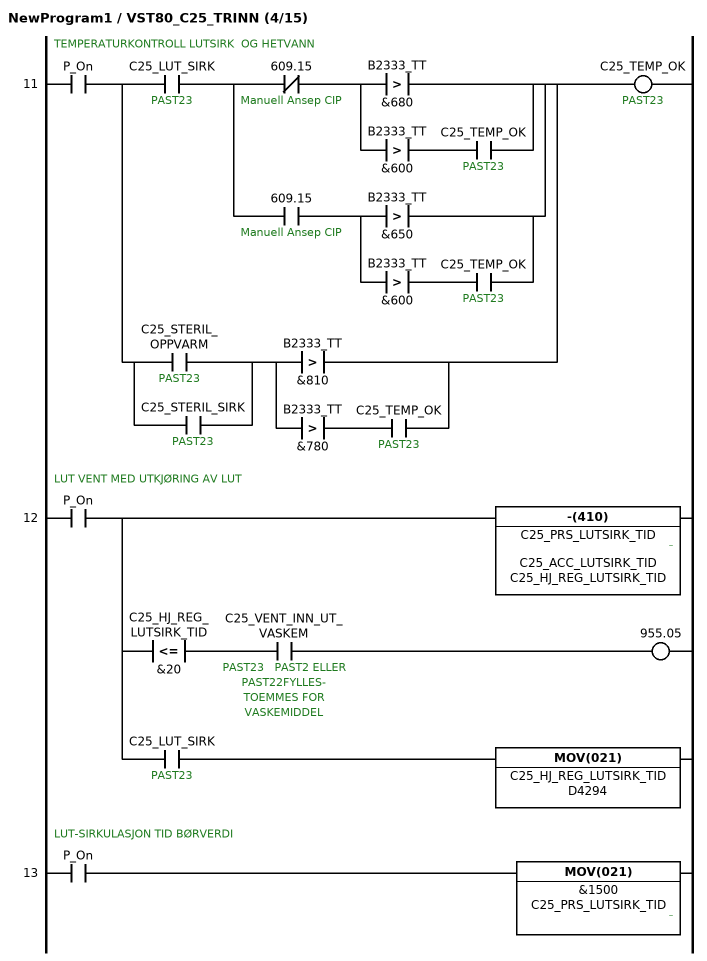
; [picture p456: NewProgram1 / VST80_C25_TRINN, rungs 11-13]
; rung 11: TEMPERATURKONTROLL LUTSIRK  OG HETVANN
LD P_On
LD C25_LUT_SIRK  ; PAST23
LDNOT 609.15  ; Manuell Ansep CIP
LD>(320) B2333_TT &680
LD>(320) B2333_TT &600
AND C25_TEMP_OK  ; PAST23
ORLD
ANDLD
LD 609.15  ; Manuell Ansep CIP
LD>(320) B2333_TT &650
LD>(320) B2333_TT &600
AND C25_TEMP_OK  ; PAST23
ORLD
ANDLD
ORLD
ANDLD
LD C25_STERIL_OPPVARM  ; PAST23
OR C25_STERIL_SIRK  ; PAST23
LD>(320) B2333_TT &810
LD>(320) B2333_TT &780
AND C25_TEMP_OK  ; PAST23
ORLD
ANDLD
ORLD
ANDLD
OUT C25_TEMP_OK  ; PAST23
; rung 12: LUT VENT MED UTKJØRING AV LUT
LD P_On
OUT TR0
-(410) C25_PRS_LUTSIRK_TID C25_ACC_LUTSIRK_TID C25_HJ_REG_LUTSIRK_TID  ; ¨
AND<=(315) C25_HJ_REG_LUTSIRK_TID &20
AND C25_VENT_INN_UT_VASKEM  ; PAST23   PAST2 ELLER PAST22FYLLES-TOEMMES FOR VASKEMIDDEL
OUT 955.05
LD TR0
AND C25_LUT_SIRK  ; PAST23
MOV(021) C25_HJ_REG_LUTSIRK_TID D4294
; rung 13: LUT-SIRKULASJON TID BØRVERDI
LD P_On
MOV(021) &1500 C25_PRS_LUTSIRK_TID  ; ¨

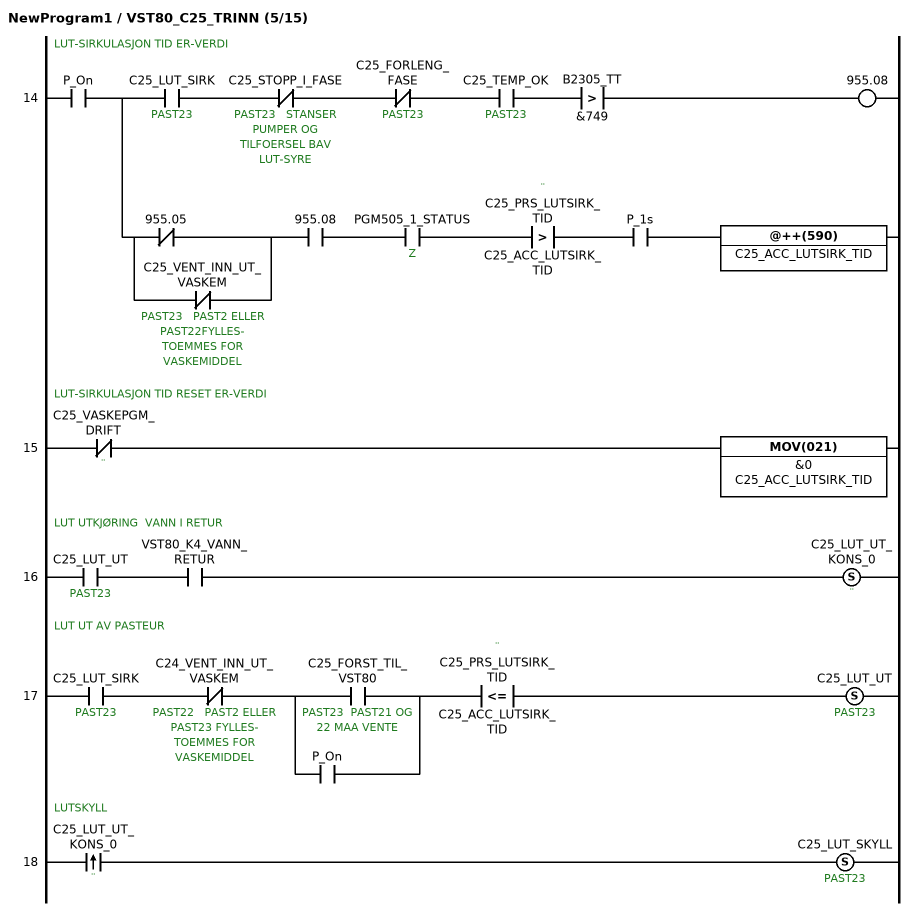
; rung 14: LUT-SIRKULASJON TID ER-VERDI
LD P_On
OUT TR0
AND C25_LUT_SIRK  ; PAST23
ANDNOT C25_STOPP_I_FASE  ; PAST23   STANSER PUMPER OG TILFOERSEL BAV LUT-SYRE
ANDNOT C25_FORLENG_FASE  ; PAST23
AND C25_TEMP_OK  ; PAST23
AND>(320) B2305_TT &749
OUT 955.08
LD TR0
LDNOT 955.05
ORNOT C25_VENT_INN_UT_VASKEM  ; PAST23   PAST2 ELLER PAST22FYLLES-TOEMMES FOR VASKEMIDDEL
ANDLD
AND 955.08
AND PGM505_1_STATUS  ; Z
AND>(320) C25_PRS_LUTSIRK_TID C25_ACC_LUTSIRK_TID  ; ¨
AND P_1s
@++(590) C25_ACC_LUTSIRK_TID
; rung 15: LUT-SIRKULASJON TID RESET ER-VERDI
LDNOT C25_VASKEPGM_DRIFT  ; ¨
MOV(021) &0 C25_ACC_LUTSIRK_TID
; rung 16: LUT UTKJØRING  VANN I RETUR
LD C25_LUT_UT  ; PAST23
AND VST80_K4_VANN_RETUR
SET C25_LUT_UT_KONS_0  ; ¨
; rung 17: LUT UT AV PASTEUR
LD C25_LUT_SIRK  ; PAST23
ANDNOT C24_VENT_INN_UT_VASKEM  ; PAST22   PAST2 ELLER PAST23 FYLLES-TOEMMES FOR VASKEMIDDEL
LD C25_FORST_TIL_VST80  ; PAST23  PAST21 OG 22 MAA VENTE
OR P_On
ANDLD
AND<=(315) C25_PRS_LUTSIRK_TID C25_ACC_LUTSIRK_TID  ; ¨
SET C25_LUT_UT  ; PAST23
; rung 18: LUTSKYLL
@LD C25_LUT_UT_KONS_0  ; ¨
SET C25_LUT_SKYLL  ; PAST23

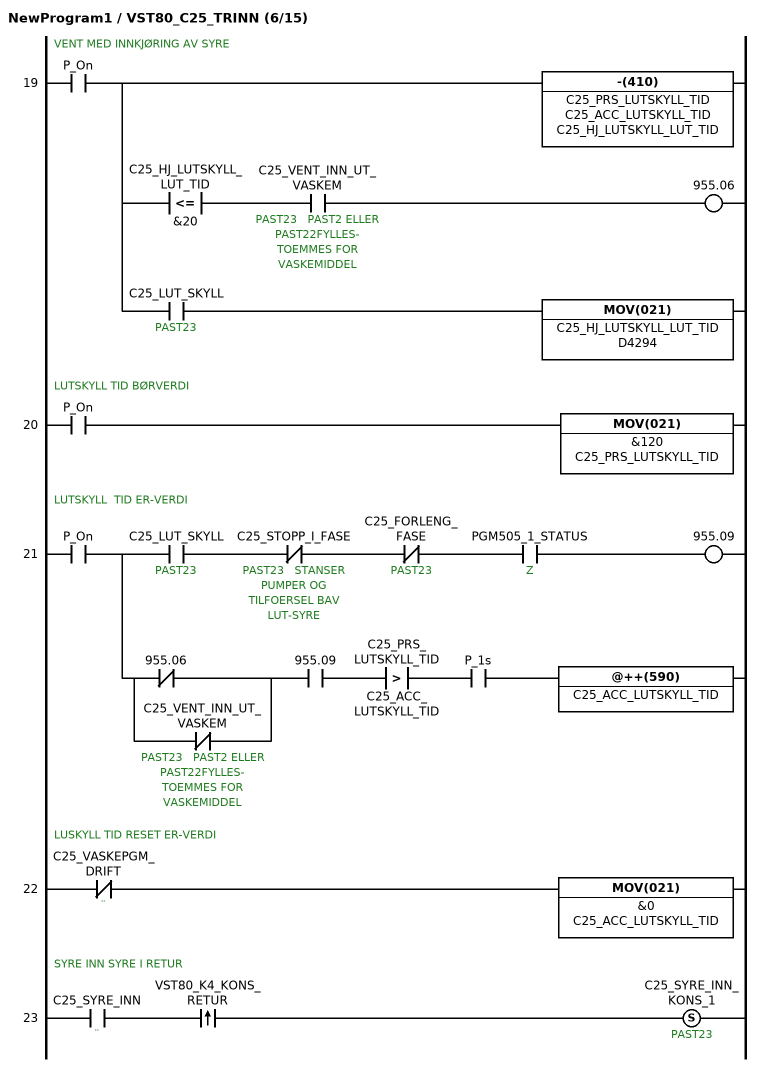
; rung 19: VENT MED INNKJØRING AV SYRE
LD P_On
OUT TR0
-(410) C25_PRS_LUTSKYLL_TID C25_ACC_LUTSKYLL_TID C25_HJ_LUTSKYLL_LUT_TID
AND<=(315) C25_HJ_LUTSKYLL_LUT_TID &20
AND C25_VENT_INN_UT_VASKEM  ; PAST23   PAST2 ELLER PAST22FYLLES-TOEMMES FOR VASKEMIDDEL
OUT 955.06
LD TR0
AND C25_LUT_SKYLL  ; PAST23
MOV(021) C25_HJ_LUTSKYLL_LUT_TID D4294
; rung 20: LUTSKYLL TID BØRVERDI
LD P_On
MOV(021) &120 C25_PRS_LUTSKYLL_TID
; rung 21: LUTSKYLL  TID ER-VERDI
LD P_On
OUT TR0
AND C25_LUT_SKYLL  ; PAST23
ANDNOT C25_STOPP_I_FASE  ; PAST23   STANSER PUMPER OG TILFOERSEL BAV LUT-SYRE
ANDNOT C25_FORLENG_FASE  ; PAST23
AND PGM505_1_STATUS  ; Z
OUT 955.09
LD TR0
LDNOT 955.06
ORNOT C25_VENT_INN_UT_VASKEM  ; PAST23   PAST2 ELLER PAST22FYLLES-TOEMMES FOR VASKEMIDDEL
ANDLD
AND 955.09
AND>(320) C25_PRS_LUTSKYLL_TID C25_ACC_LUTSKYLL_TID
AND P_1s
@++(590) C25_ACC_LUTSKYLL_TID
; rung 22: LUSKYLL TID RESET ER-VERDI
LDNOT C25_VASKEPGM_DRIFT  ; ¨
MOV(021) &0 C25_ACC_LUTSKYLL_TID
; rung 23: SYRE INN SYRE I RETUR
LD C25_SYRE_INN  ; ¨
@AND VST80_K4_KONS_RETUR
SET C25_SYRE_INN_KONS_1  ; PAST23

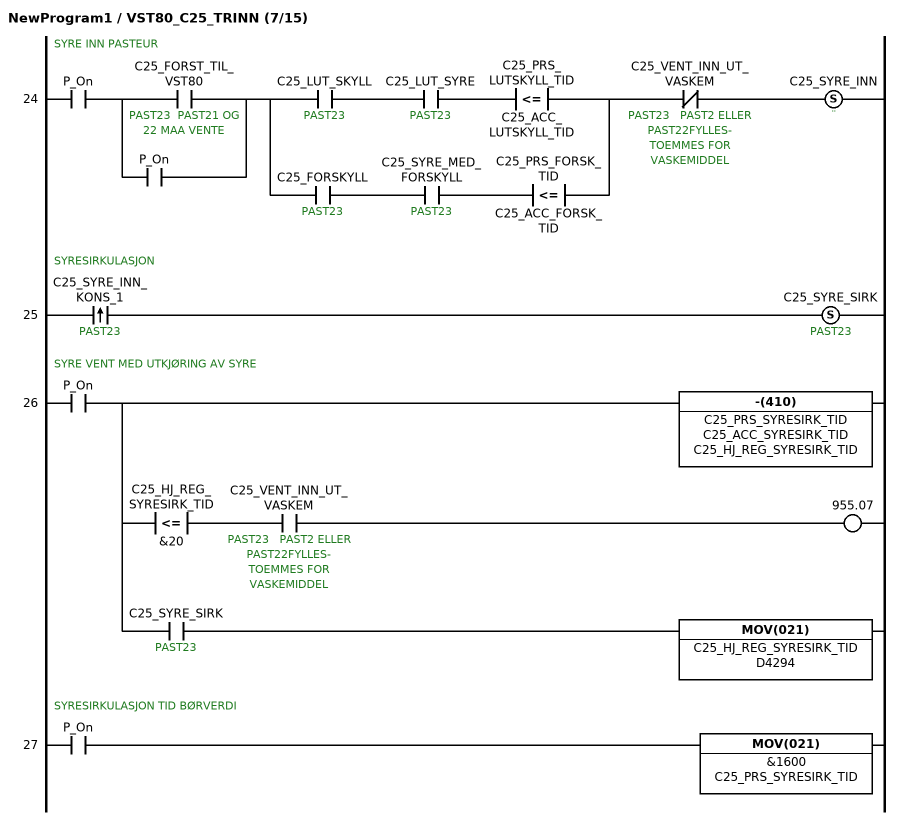
; rung 24: SYRE INN PASTEUR
LD P_On
LD C25_FORST_TIL_VST80  ; PAST23  PAST21 OG 22 MAA VENTE
OR P_On
ANDLD
LD C25_LUT_SKYLL  ; PAST23
AND C25_LUT_SYRE  ; PAST23
AND<=(315) C25_PRS_LUTSKYLL_TID C25_ACC_LUTSKYLL_TID
LD C25_FORSKYLL  ; PAST23
AND C25_SYRE_MED_FORSKYLL  ; PAST23
AND<=(315) C25_PRS_FORSK_TID C25_ACC_FORSK_TID
ORLD
ANDLD
ANDNOT C25_VENT_INN_UT_VASKEM  ; PAST23   PAST2 ELLER PAST22FYLLES-TOEMMES FOR VASKEMIDDEL
SET C25_SYRE_INN  ; ¨
; rung 25: SYRESIRKULASJON
@LD C25_SYRE_INN_KONS_1  ; PAST23
SET C25_SYRE_SIRK  ; PAST23
; rung 26: SYRE VENT MED UTKJØRING AV SYRE
LD P_On
OUT TR0
-(410) C25_PRS_SYRESIRK_TID C25_ACC_SYRESIRK_TID C25_HJ_REG_SYRESIRK_TID
AND<=(315) C25_HJ_REG_SYRESIRK_TID &20
AND C25_VENT_INN_UT_VASKEM  ; PAST23   PAST2 ELLER PAST22FYLLES-TOEMMES FOR VASKEMIDDEL
OUT 955.07
LD TR0
AND C25_SYRE_SIRK  ; PAST23
MOV(021) C25_HJ_REG_SYRESIRK_TID D4294
; rung 27: SYRESIRKULASJON TID BØRVERDI
LD P_On
MOV(021) &1600 C25_PRS_SYRESIRK_TID

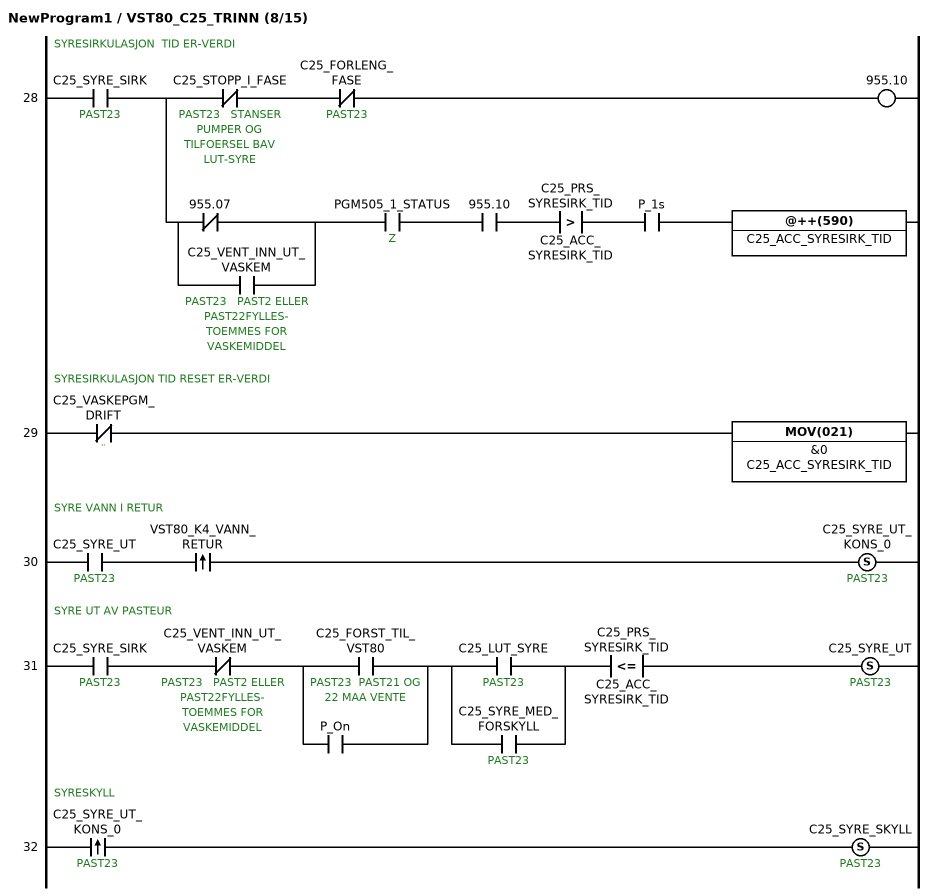
; rung 28: SYRESIRKULASJON  TID ER-VERDI
LD C25_SYRE_SIRK  ; PAST23
OUT TR0
ANDNOT C25_STOPP_I_FASE  ; PAST23   STANSER PUMPER OG TILFOERSEL BAV LUT-SYRE
ANDNOT C25_FORLENG_FASE  ; PAST23
OUT 955.10
LD TR0
LDNOT 955.07
OR C25_VENT_INN_UT_VASKEM  ; PAST23   PAST2 ELLER PAST22FYLLES-TOEMMES FOR VASKEMIDDEL
ANDLD
AND PGM505_1_STATUS  ; Z
AND 955.10
AND>(320) C25_PRS_SYRESIRK_TID C25_ACC_SYRESIRK_TID
AND P_1s
@++(590) C25_ACC_SYRESIRK_TID
; rung 29: SYRESIRKULASJON TID RESET ER-VERDI
LDNOT C25_VASKEPGM_DRIFT  ; ¨
MOV(021) &0 C25_ACC_SYRESIRK_TID
; rung 30: SYRE VANN I RETUR
LD C25_SYRE_UT  ; PAST23
@AND VST80_K4_VANN_RETUR
SET C25_SYRE_UT_KONS_0  ; PAST23
; rung 31: SYRE UT AV PASTEUR
LD C25_SYRE_SIRK  ; PAST23
ANDNOT C25_VENT_INN_UT_VASKEM  ; PAST23   PAST2 ELLER PAST22FYLLES-TOEMMES FOR VASKEMIDDEL
LD C25_FORST_TIL_VST80  ; PAST23  PAST21 OG 22 MAA VENTE
OR P_On
ANDLD
LD C25_LUT_SYRE  ; PAST23
OR C25_SYRE_MED_FORSKYLL  ; PAST23
ANDLD
AND<=(315) C25_PRS_SYRESIRK_TID C25_ACC_SYRESIRK_TID
SET C25_SYRE_UT  ; PAST23
; rung 32: SYRESKYLL
@LD C25_SYRE_UT_KONS_0  ; PAST23
SET C25_SYRE_SKYLL  ; PAST23

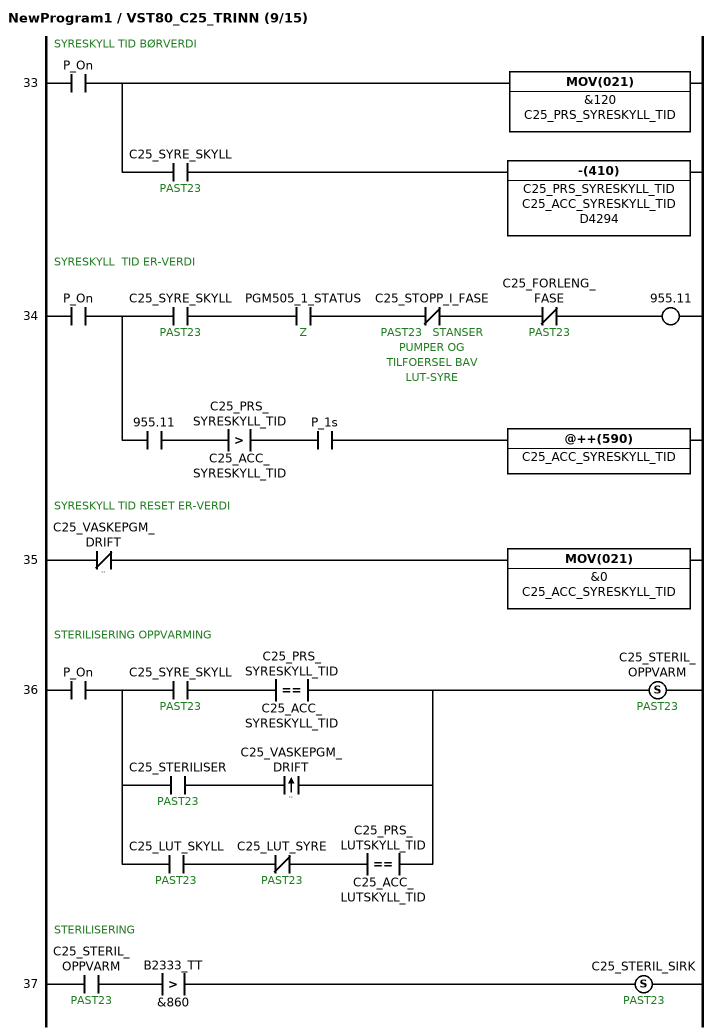
; rung 33: SYRESKYLL TID BØRVERDI
LD P_On
MOV(021) &120 C25_PRS_SYRESKYLL_TID
AND C25_SYRE_SKYLL  ; PAST23
-(410) C25_PRS_SYRESKYLL_TID C25_ACC_SYRESKYLL_TID D4294
; rung 34: SYRESKYLL  TID ER-VERDI
LD P_On
OUT TR0
AND C25_SYRE_SKYLL  ; PAST23
AND PGM505_1_STATUS  ; Z
ANDNOT C25_STOPP_I_FASE  ; PAST23   STANSER PUMPER OG TILFOERSEL BAV LUT-SYRE
ANDNOT C25_FORLENG_FASE  ; PAST23
OUT 955.11
LD TR0
AND 955.11
AND>(320) C25_PRS_SYRESKYLL_TID C25_ACC_SYRESKYLL_TID
AND P_1s
@++(590) C25_ACC_SYRESKYLL_TID
; rung 35: SYRESKYLL TID RESET ER-VERDI
LDNOT C25_VASKEPGM_DRIFT  ; ¨
MOV(021) &0 C25_ACC_SYRESKYLL_TID
; rung 36: STERILISERING OPPVARMING
LD P_On
LD C25_SYRE_SKYLL  ; PAST23
AND=(300) C25_PRS_SYRESKYLL_TID C25_ACC_SYRESKYLL_TID
LD C25_STERILISER  ; PAST23
@AND C25_VASKEPGM_DRIFT  ; ¨
ORLD
LD C25_LUT_SKYLL  ; PAST23
ANDNOT C25_LUT_SYRE  ; PAST23
AND=(300) C25_PRS_LUTSKYLL_TID C25_ACC_LUTSKYLL_TID
ORLD
ANDLD
SET C25_STERIL_OPPVARM  ; PAST23
; rung 37: STERILISERING
LD C25_STERIL_OPPVARM  ; PAST23
AND>(320) B2333_TT &860
SET C25_STERIL_SIRK  ; PAST23

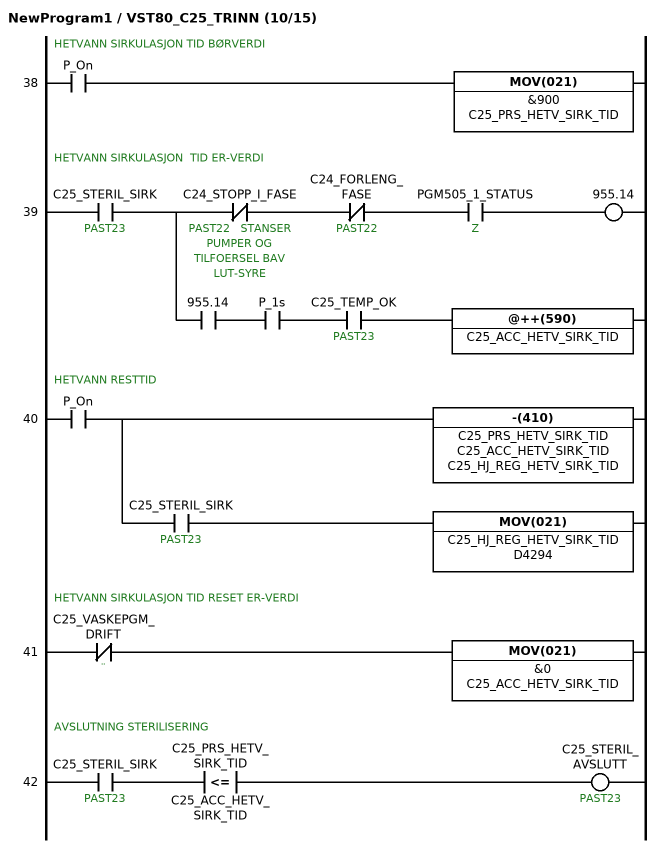
; rung 38: HETVANN SIRKULASJON TID BØRVERDI
LD P_On
MOV(021) &900 C25_PRS_HETV_SIRK_TID
; rung 39: HETVANN SIRKULASJON  TID ER-VERDI
LD C25_STERIL_SIRK  ; PAST23
OUT TR0
ANDNOT C24_STOPP_I_FASE  ; PAST22   STANSER PUMPER OG TILFOERSEL BAV LUT-SYRE
ANDNOT C24_FORLENG_FASE  ; PAST22
AND PGM505_1_STATUS  ; Z
OUT 955.14
LD TR0
AND 955.14
AND P_1s
AND C25_TEMP_OK  ; PAST23
@++(590) C25_ACC_HETV_SIRK_TID
; rung 40: HETVANN RESTTID
LD P_On
-(410) C25_PRS_HETV_SIRK_TID C25_ACC_HETV_SIRK_TID C25_HJ_REG_HETV_SIRK_TID
AND C25_STERIL_SIRK  ; PAST23
MOV(021) C25_HJ_REG_HETV_SIRK_TID D4294
; rung 41: HETVANN SIRKULASJON TID RESET ER-VERDI
LDNOT C25_VASKEPGM_DRIFT  ; ¨
MOV(021) &0 C25_ACC_HETV_SIRK_TID
; rung 42: AVSLUTNING STERILISERING
LD C25_STERIL_SIRK  ; PAST23
AND<=(315) C25_PRS_HETV_SIRK_TID C25_ACC_HETV_SIRK_TID
OUT C25_STERIL_AVSLUTT  ; PAST23

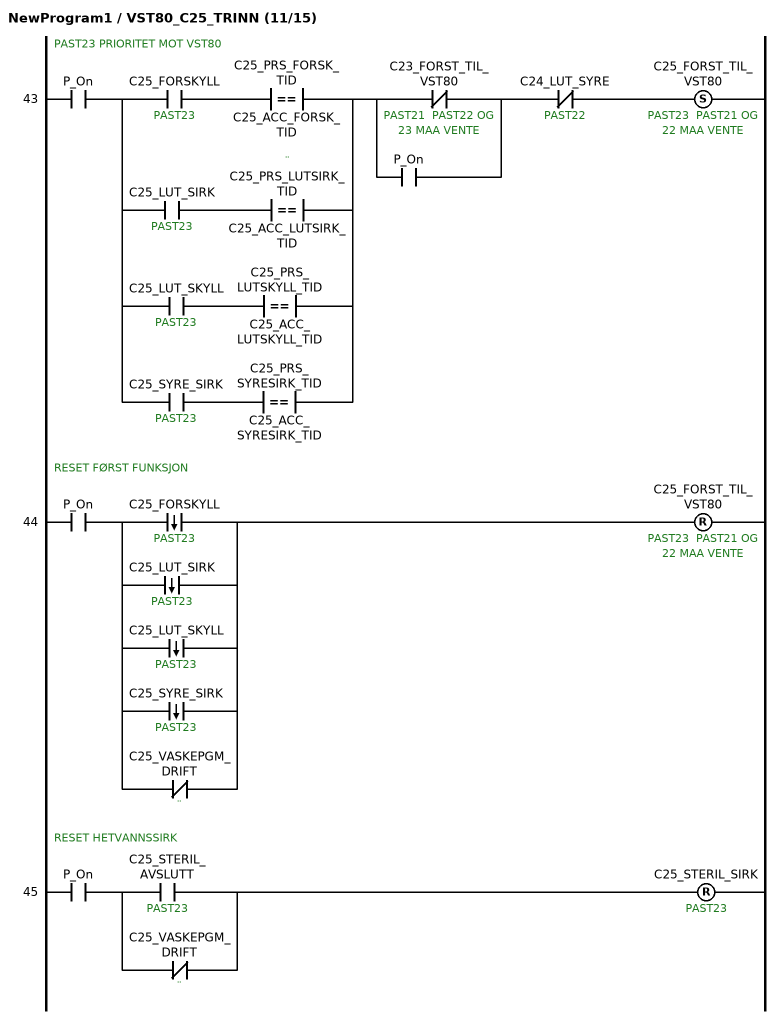
; rung 43: PAST23 PRIORITET MOT VST80
LD P_On
LD C25_FORSKYLL  ; PAST23
AND=(300) C25_PRS_FORSK_TID C25_ACC_FORSK_TID
LD C25_LUT_SIRK  ; PAST23
AND=(300) C25_PRS_LUTSIRK_TID C25_ACC_LUTSIRK_TID  ; ¨
ORLD
LD C25_LUT_SKYLL  ; PAST23
AND=(300) C25_PRS_LUTSKYLL_TID C25_ACC_LUTSKYLL_TID
ORLD
LD C25_SYRE_SIRK  ; PAST23
AND=(300) C25_PRS_SYRESIRK_TID C25_ACC_SYRESIRK_TID
ORLD
ANDLD
LDNOT C23_FORST_TIL_VST80  ; PAST21  PAST22 OG 23 MAA VENTE
OR P_On
ANDLD
ANDNOT C24_LUT_SYRE  ; PAST22
SET C25_FORST_TIL_VST80  ; PAST23  PAST21 OG 22 MAA VENTE
; rung 44: RESET FØRST FUNKSJON
LD P_On
%LD C25_FORSKYLL  ; PAST23
%OR C25_LUT_SIRK  ; PAST23
%OR C25_LUT_SKYLL  ; PAST23
%OR C25_SYRE_SIRK  ; PAST23
ORNOT C25_VASKEPGM_DRIFT  ; ¨
ANDLD
RSET C25_FORST_TIL_VST80  ; PAST23  PAST21 OG 22 MAA VENTE
; rung 45: RESET HETVANNSSIRK
LD P_On
LD C25_STERIL_AVSLUTT  ; PAST23
ORNOT C25_VASKEPGM_DRIFT  ; ¨
ANDLD
RSET C25_STERIL_SIRK  ; PAST23

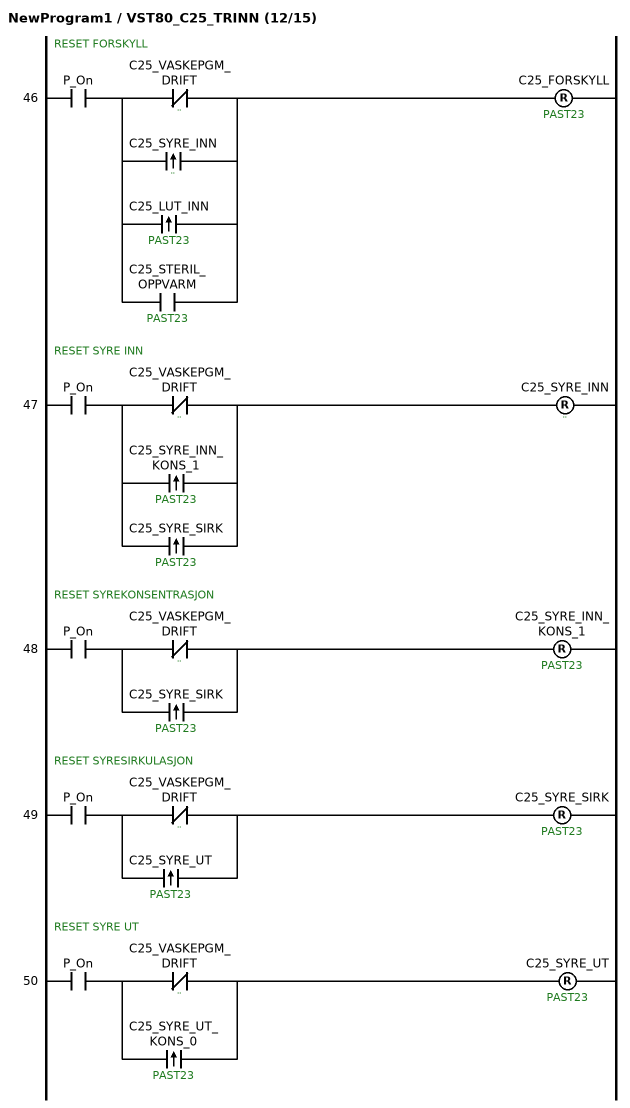
; rung 46: RESET FORSKYLL
LD P_On
LDNOT C25_VASKEPGM_DRIFT  ; ¨
@OR C25_SYRE_INN  ; ¨
@OR C25_LUT_INN  ; PAST23
OR C25_STERIL_OPPVARM  ; PAST23
ANDLD
RSET C25_FORSKYLL  ; PAST23
; rung 47: RESET SYRE INN
LD P_On
LDNOT C25_VASKEPGM_DRIFT  ; ¨
@OR C25_SYRE_INN_KONS_1  ; PAST23
@OR C25_SYRE_SIRK  ; PAST23
ANDLD
RSET C25_SYRE_INN  ; ¨
; rung 48: RESET SYREKONSENTRASJON
LD P_On
LDNOT C25_VASKEPGM_DRIFT  ; ¨
@OR C25_SYRE_SIRK  ; PAST23
ANDLD
RSET C25_SYRE_INN_KONS_1  ; PAST23
; rung 49: RESET SYRESIRKULASJON
LD P_On
LDNOT C25_VASKEPGM_DRIFT  ; ¨
@OR C25_SYRE_UT  ; PAST23
ANDLD
RSET C25_SYRE_SIRK  ; PAST23
; rung 50: RESET SYRE UT
LD P_On
LDNOT C25_VASKEPGM_DRIFT  ; ¨
@OR C25_SYRE_UT_KONS_0  ; PAST23
ANDLD
RSET C25_SYRE_UT  ; PAST23

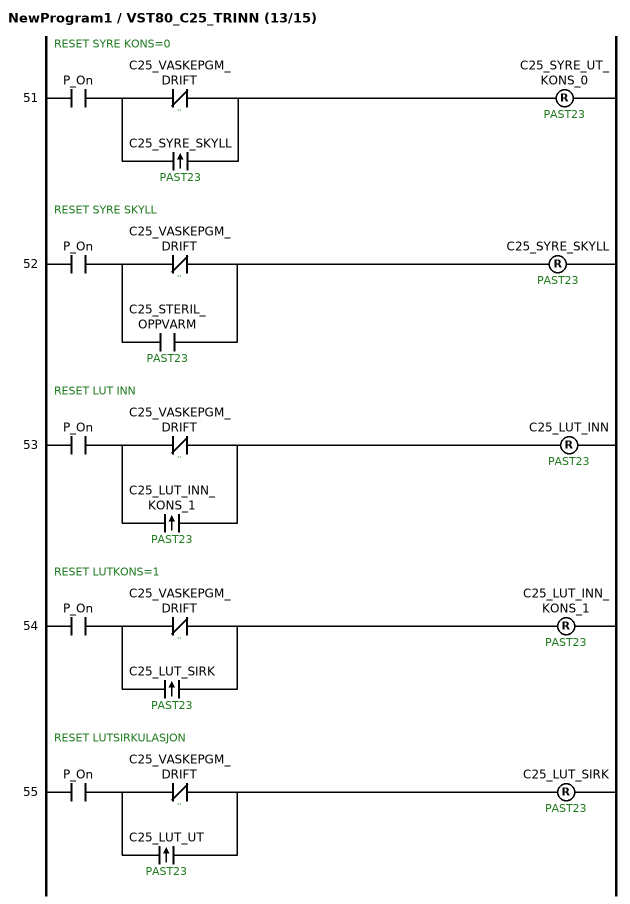
; rung 51: RESET SYRE KONS=0
LD P_On
LDNOT C25_VASKEPGM_DRIFT  ; ¨
@OR C25_SYRE_SKYLL  ; PAST23
ANDLD
RSET C25_SYRE_UT_KONS_0  ; PAST23
; rung 52: RESET SYRE SKYLL
LD P_On
LDNOT C25_VASKEPGM_DRIFT  ; ¨
OR C25_STERIL_OPPVARM  ; PAST23
ANDLD
RSET C25_SYRE_SKYLL  ; PAST23
; rung 53: RESET LUT INN
LD P_On
LDNOT C25_VASKEPGM_DRIFT  ; ¨
@OR C25_LUT_INN_KONS_1  ; PAST23
ANDLD
RSET C25_LUT_INN  ; PAST23
; rung 54: RESET LUTKONS=1
LD P_On
LDNOT C25_VASKEPGM_DRIFT  ; ¨
@OR C25_LUT_SIRK  ; PAST23
ANDLD
RSET C25_LUT_INN_KONS_1  ; PAST23
; rung 55: RESET LUTSIRKULASJON
LD P_On
LDNOT C25_VASKEPGM_DRIFT  ; ¨
@OR C25_LUT_UT  ; PAST23
ANDLD
RSET C25_LUT_SIRK  ; PAST23

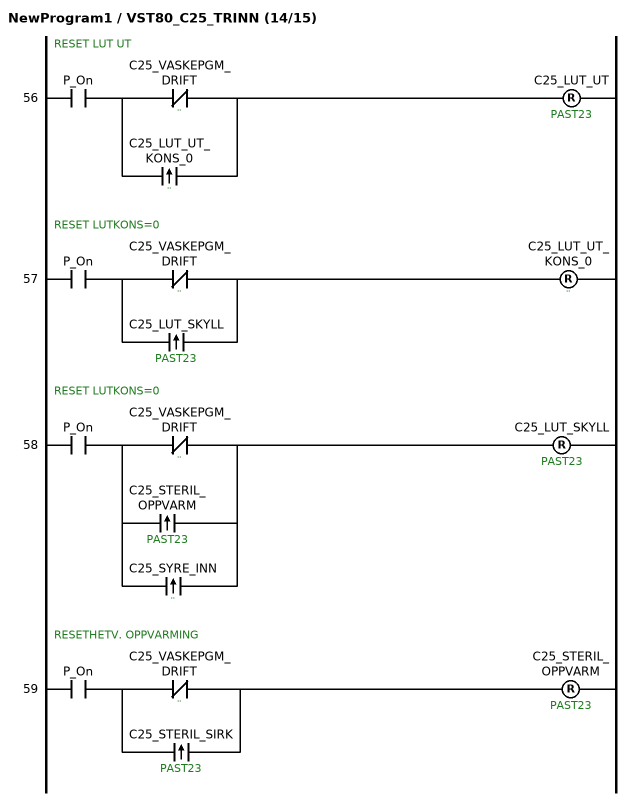
; rung 56: RESET LUT UT
LD P_On
LDNOT C25_VASKEPGM_DRIFT  ; ¨
@OR C25_LUT_UT_KONS_0  ; ¨
ANDLD
RSET C25_LUT_UT  ; PAST23
; rung 57: RESET LUTKONS=0
LD P_On
LDNOT C25_VASKEPGM_DRIFT  ; ¨
@OR C25_LUT_SKYLL  ; PAST23
ANDLD
RSET C25_LUT_UT_KONS_0  ; ¨
; rung 58: RESET LUTKONS=0
LD P_On
LDNOT C25_VASKEPGM_DRIFT  ; ¨
@OR C25_STERIL_OPPVARM  ; PAST23
@OR C25_SYRE_INN  ; ¨
ANDLD
RSET C25_LUT_SKYLL  ; PAST23
; rung 59: RESETHETV. OPPVARMING
LD P_On
LDNOT C25_VASKEPGM_DRIFT  ; ¨
@OR C25_STERIL_SIRK  ; PAST23
ANDLD
RSET C25_STERIL_OPPVARM  ; PAST23

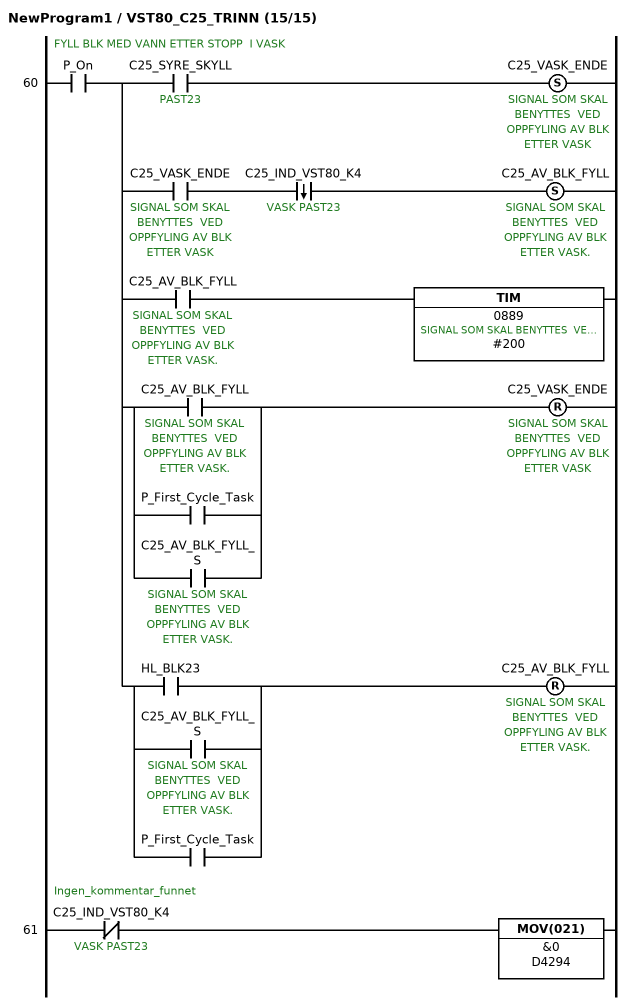
; rung 60: FYLL BLK MED VANN ETTER STOPP  I VASK
LD P_On
OUT TR0
AND C25_SYRE_SKYLL  ; PAST23
SET C25_VASK_ENDE  ; SIGNAL SOM SKAL BENYTTES  VED OPPFYLING AV BLK ETTER VASK
LD TR0
AND C25_VASK_ENDE  ; SIGNAL SOM SKAL BENYTTES  VED OPPFYLING AV BLK ETTER VASK
%AND C25_IND_VST80_K4  ; VASK PAST23
SET C25_AV_BLK_FYLL  ; SIGNAL SOM SKAL BENYTTES  VED OPPFYLING AV BLK ETTER VASK.
LD TR0
AND C25_AV_BLK_FYLL  ; SIGNAL SOM SKAL BENYTTES  VED OPPFYLING AV BLK ETTER VASK.
TIM 0889 #200  ; SIGNAL SOM SKAL BENYTTES  VED OPPFYLING AV BLK ETTER VASK.
LD TR0
LD C25_AV_BLK_FYLL  ; SIGNAL SOM SKAL BENYTTES  VED OPPFYLING AV BLK ETTER VASK.
OR P_First_Cycle_Task
OR C25_AV_BLK_FYLL_S  ; SIGNAL SOM SKAL BENYTTES  VED OPPFYLING AV BLK ETTER VASK.
ANDLD
RSET C25_VASK_ENDE  ; SIGNAL SOM SKAL BENYTTES  VED OPPFYLING AV BLK ETTER VASK
LD TR0
LD HL_BLK23
OR C25_AV_BLK_FYLL_S  ; SIGNAL SOM SKAL BENYTTES  VED OPPFYLING AV BLK ETTER VASK.
OR P_First_Cycle_Task
ANDLD
RSET C25_AV_BLK_FYLL  ; SIGNAL SOM SKAL BENYTTES  VED OPPFYLING AV BLK ETTER VASK.
; rung 61: Ingen_kommentar_funnet
LDNOT C25_IND_VST80_K4  ; VASK PAST23
MOV(021) &0 D4294
; rung 62: Ingen_kommentar_funnet

### Section VST80_C25_GRAFIKK_TEKSTER

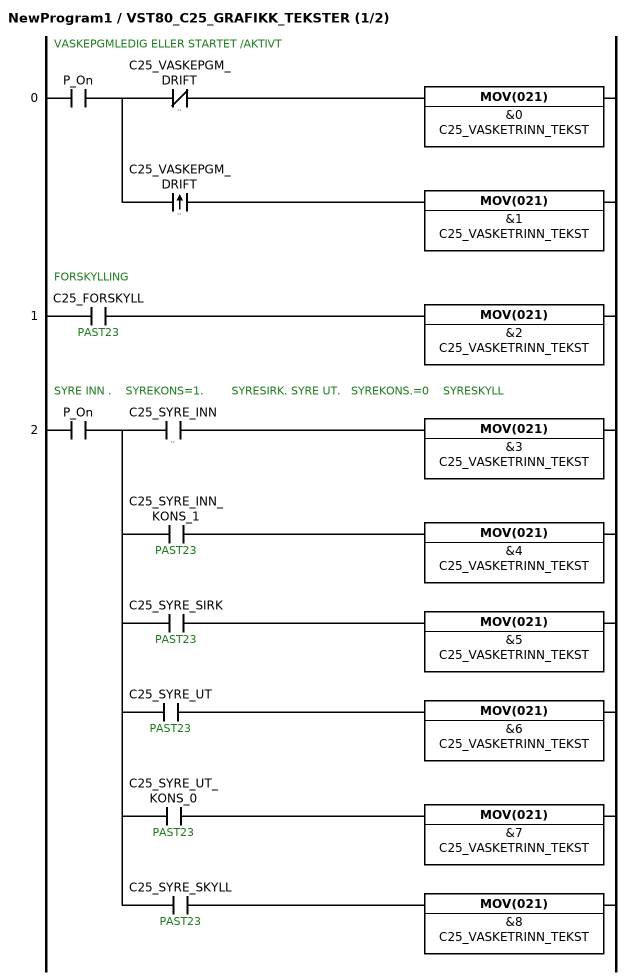
; rung 0: VASKEPGMLEDIG ELLER STARTET /AKTIVT
LD P_On
OUT TR0
ANDNOT C25_VASKEPGM_DRIFT  ; ¨
MOV(021) &0 C25_VASKETRINN_TEKST
LD TR0
@AND C25_VASKEPGM_DRIFT  ; ¨
MOV(021) &1 C25_VASKETRINN_TEKST
; rung 1: FORSKYLLING
LD C25_FORSKYLL  ; PAST23
MOV(021) &2 C25_VASKETRINN_TEKST
; rung 2: SYRE INN .    SYREKONS=1.        SYRESIRK. SYRE UT.   SYREKONS.=0    SYRESKYLL
LD P_On
OUT TR0
AND C25_SYRE_INN  ; ¨
MOV(021) &3 C25_VASKETRINN_TEKST
LD TR0
AND C25_SYRE_INN_KONS_1  ; PAST23
MOV(021) &4 C25_VASKETRINN_TEKST
LD TR0
AND C25_SYRE_SIRK  ; PAST23
MOV(021) &5 C25_VASKETRINN_TEKST
LD TR0
AND C25_SYRE_UT  ; PAST23
MOV(021) &6 C25_VASKETRINN_TEKST
LD TR0
AND C25_SYRE_UT_KONS_0  ; PAST23
MOV(021) &7 C25_VASKETRINN_TEKST
LD TR0
AND C25_SYRE_SKYLL  ; PAST23
MOV(021) &8 C25_VASKETRINN_TEKST

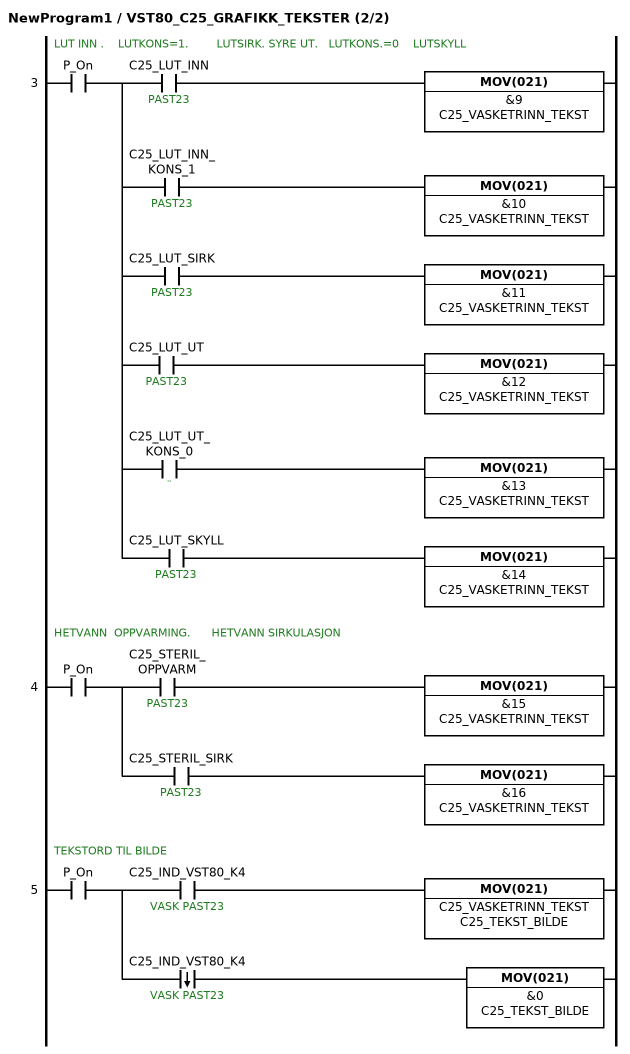
; rung 3: LUT INN .    LUTKONS=1.        LUTSIRK. SYRE UT.   LUTKONS.=0    LUTSKYLL
LD P_On
OUT TR0
AND C25_LUT_INN  ; PAST23
MOV(021) &9 C25_VASKETRINN_TEKST
LD TR0
AND C25_LUT_INN_KONS_1  ; PAST23
MOV(021) &10 C25_VASKETRINN_TEKST
LD TR0
AND C25_LUT_SIRK  ; PAST23
MOV(021) &11 C25_VASKETRINN_TEKST
LD TR0
AND C25_LUT_UT  ; PAST23
MOV(021) &12 C25_VASKETRINN_TEKST
LD TR0
AND C25_LUT_UT_KONS_0  ; ¨
MOV(021) &13 C25_VASKETRINN_TEKST
LD TR0
AND C25_LUT_SKYLL  ; PAST23
MOV(021) &14 C25_VASKETRINN_TEKST
; rung 4: HETVANN  OPPVARMING.      HETVANN SIRKULASJON
LD P_On
OUT TR0
AND C25_STERIL_OPPVARM  ; PAST23
MOV(021) &15 C25_VASKETRINN_TEKST
LD TR0
AND C25_STERIL_SIRK  ; PAST23
MOV(021) &16 C25_VASKETRINN_TEKST
; rung 5: TEKSTORD TIL BILDE
LD P_On
OUT TR0
AND C25_IND_VST80_K4  ; VASK PAST23
MOV(021) C25_VASKETRINN_TEKST C25_TEKST_BILDE
LD TR0
%AND C25_IND_VST80_K4  ; VASK PAST23
MOV(021) &0 C25_TEKST_BILDE
; rung 6: Ingen_kommentar_funnet

### Section C25_VASKERAPPORT

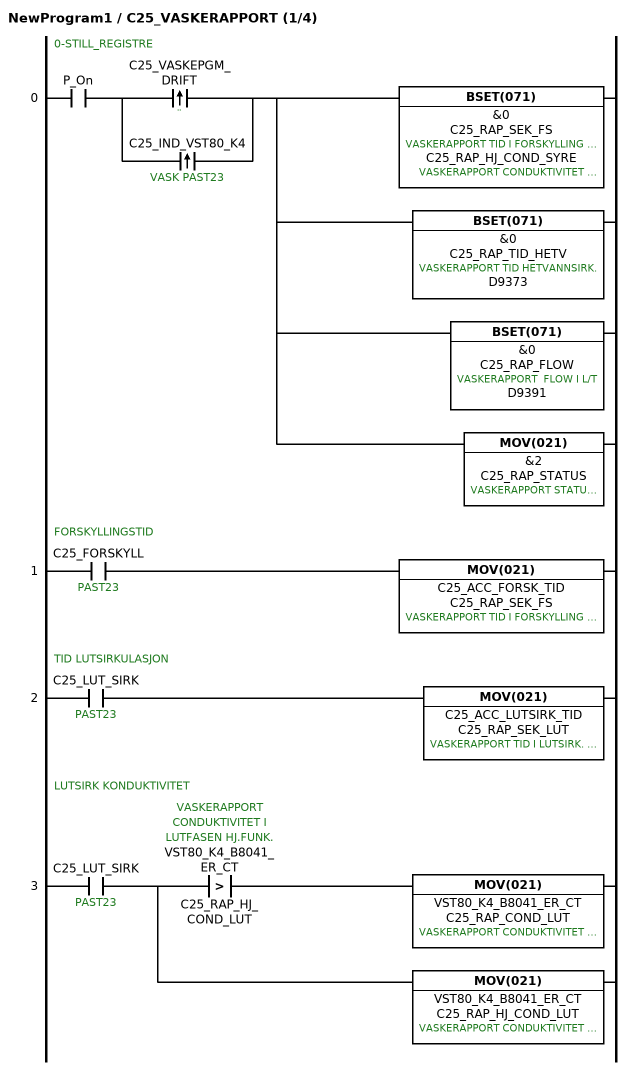
; rung 0: 0-STILL_REGISTRE
LD P_On
@LD C25_VASKEPGM_DRIFT  ; ¨
@OR C25_IND_VST80_K4  ; VASK PAST23
ANDLD
BSET(071) &0 C25_RAP_SEK_FS C25_RAP_HJ_COND_SYRE  ; VASKERAPPORT TID I FORSKYLLING I SEKUNDER, VASKERAPPORT CONDUKTIVITET I SYREFASEN HJ.FUNK.
BSET(071) &0 C25_RAP_TID_HETV D9373  ; VASKERAPPORT TID HETVANNSIRK.
BSET(071) &0 C25_RAP_FLOW D9391  ; VASKERAPPORT  FLOW I L/T
MOV(021) &2 C25_RAP_STATUS  ; VASKERAPPORT STATUS          0=GODKJ.  1=DRIFTFORS.  2= IKKE GODKJ.
; rung 1: FORSKYLLINGSTID
LD C25_FORSKYLL  ; PAST23
MOV(021) C25_ACC_FORSK_TID C25_RAP_SEK_FS  ; VASKERAPPORT TID I FORSKYLLING I SEKUNDER
; rung 2: TID LUTSIRKULASJON
LD C25_LUT_SIRK  ; PAST23
MOV(021) C25_ACC_LUTSIRK_TID C25_RAP_SEK_LUT  ; VASKERAPPORT TID I LUTSIRK. I SEKUNDER
; rung 3: LUTSIRK KONDUKTIVITET
LD C25_LUT_SIRK  ; PAST23
OUT TR0
AND>(320) VST80_K4_B8041_ER_CT C25_RAP_HJ_COND_LUT  ; VASKERAPPORT CONDUKTIVITET I LUTFASEN HJ.FUNK.
MOV(021) VST80_K4_B8041_ER_CT C25_RAP_COND_LUT  ; VASKERAPPORT CONDUKTIVITET I LUTFASEN
LD TR0
MOV(021) VST80_K4_B8041_ER_CT C25_RAP_HJ_COND_LUT  ; VASKERAPPORT CONDUKTIVITET I LUTFASEN HJ.FUNK.

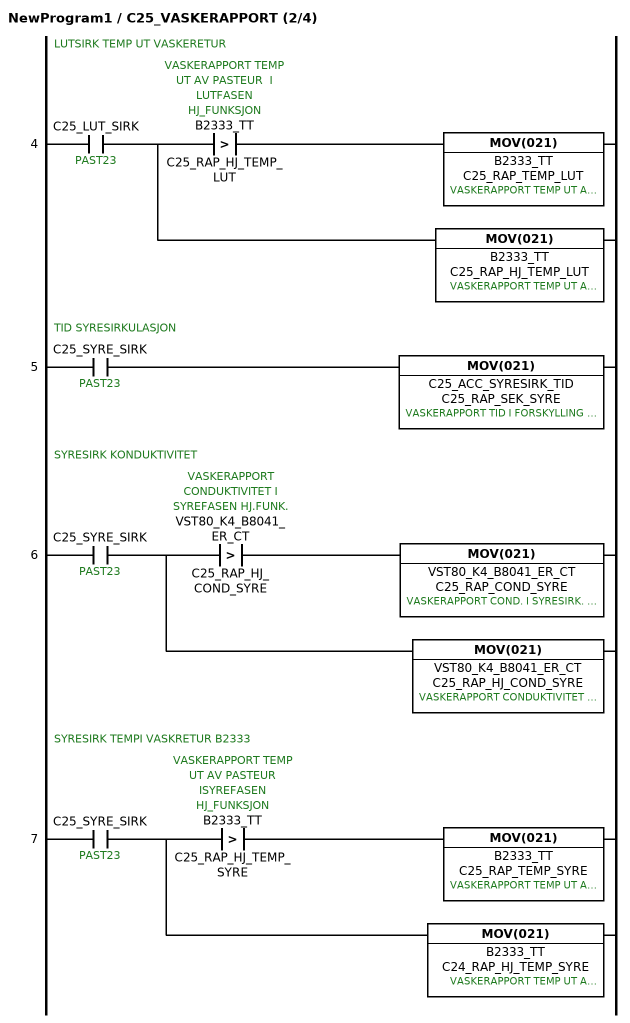
; rung 4: LUTSIRK TEMP UT VASKERETUR
LD C25_LUT_SIRK  ; PAST23
OUT TR0
AND>(320) B2333_TT C25_RAP_HJ_TEMP_LUT  ; VASKERAPPORT TEMP UT AV PASTEUR  I LUTFASEN HJ_FUNKSJON
MOV(021) B2333_TT C25_RAP_TEMP_LUT  ; VASKERAPPORT TEMP UT AV PASTEUR  I LUTFASEN
LD TR0
MOV(021) B2333_TT C25_RAP_HJ_TEMP_LUT  ; VASKERAPPORT TEMP UT AV PASTEUR  I LUTFASEN HJ_FUNKSJON
; rung 5: TID SYRESIRKULASJON
LD C25_SYRE_SIRK  ; PAST23
MOV(021) C25_ACC_SYRESIRK_TID C25_RAP_SEK_SYRE  ; VASKERAPPORT TID I FORSKYLLING I SEKUNDER
; rung 6: SYRESIRK KONDUKTIVITET
LD C25_SYRE_SIRK  ; PAST23
OUT TR0
AND>(320) VST80_K4_B8041_ER_CT C25_RAP_HJ_COND_SYRE  ; VASKERAPPORT CONDUKTIVITET I SYREFASEN HJ.FUNK.
MOV(021) VST80_K4_B8041_ER_CT C25_RAP_COND_SYRE  ; VASKERAPPORT COND. I SYRESIRK. I SEKUNDER
LD TR0
MOV(021) VST80_K4_B8041_ER_CT C25_RAP_HJ_COND_SYRE  ; VASKERAPPORT CONDUKTIVITET I SYREFASEN HJ.FUNK.
; rung 7: SYRESIRK TEMPI VASKRETUR B2333
LD C25_SYRE_SIRK  ; PAST23
OUT TR0
AND>(320) B2333_TT C25_RAP_HJ_TEMP_SYRE  ; VASKERAPPORT TEMP UT AV PASTEUR ISYREFASEN HJ_FUNKSJON
MOV(021) B2333_TT C25_RAP_TEMP_SYRE  ; VASKERAPPORT TEMP UT AV PASTEUR ISYREFASEN
LD TR0
MOV(021) B2333_TT C24_RAP_HJ_TEMP_SYRE  ; VASKERAPPORT TEMP UT AV PASTEUR ISYREFASEN HJ_FUNKSJON

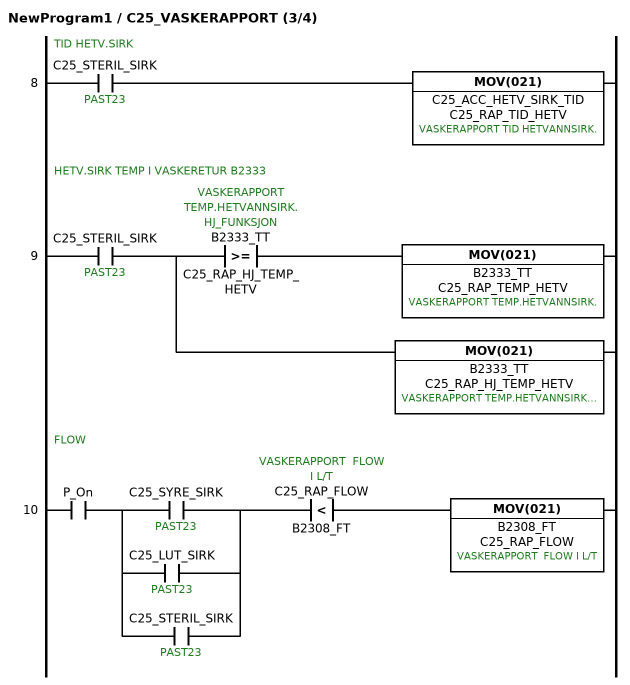
; rung 8: TID HETV.SIRK
LD C25_STERIL_SIRK  ; PAST23
MOV(021) C25_ACC_HETV_SIRK_TID C25_RAP_TID_HETV  ; VASKERAPPORT TID HETVANNSIRK.
; rung 9: HETV.SIRK TEMP I VASKERETUR B2333
LD C25_STERIL_SIRK  ; PAST23
OUT TR0
AND>=(325) B2333_TT C25_RAP_HJ_TEMP_HETV  ; VASKERAPPORT TEMP.HETVANNSIRK. HJ_FUNKSJON
MOV(021) B2333_TT C25_RAP_TEMP_HETV  ; VASKERAPPORT TEMP.HETVANNSIRK.
LD TR0
MOV(021) B2333_TT C25_RAP_HJ_TEMP_HETV  ; VASKERAPPORT TEMP.HETVANNSIRK. HJ_FUNKSJON
; rung 10: FLOW
LD P_On
LD C25_SYRE_SIRK  ; PAST23
OR C25_LUT_SIRK  ; PAST23
OR C25_STERIL_SIRK  ; PAST23
ANDLD
AND<(310) C25_RAP_FLOW B2308_FT  ; VASKERAPPORT  FLOW I L/T
MOV(021) B2308_FT C25_RAP_FLOW  ; VASKERAPPORT  FLOW I L/T

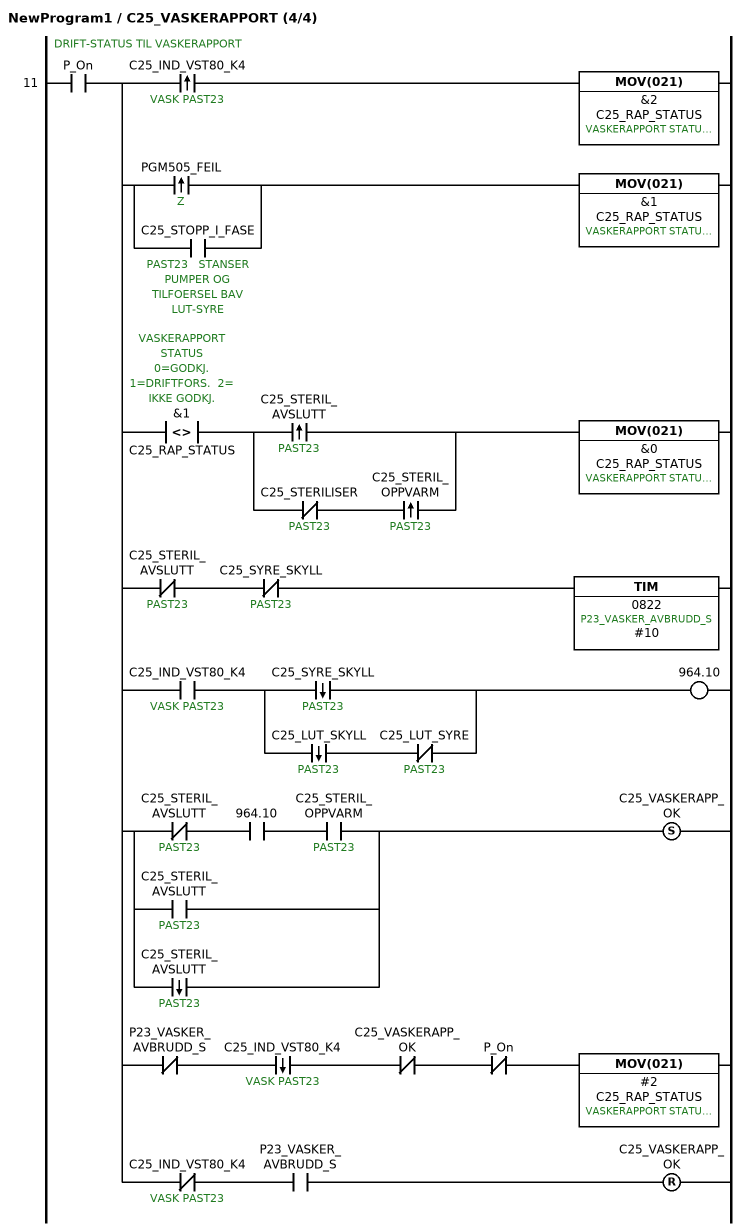
; rung 11: DRIFT-STATUS TIL VASKERAPPORT
LD P_On
OUT TR0
@AND C25_IND_VST80_K4  ; VASK PAST23
MOV(021) &2 C25_RAP_STATUS  ; VASKERAPPORT STATUS          0=GODKJ.  1=DRIFTFORS.  2= IKKE GODKJ.
LD TR0
@LD PGM505_FEIL  ; Z
OR C25_STOPP_I_FASE  ; PAST23   STANSER PUMPER OG TILFOERSEL BAV LUT-SYRE
ANDLD
MOV(021) &1 C25_RAP_STATUS  ; VASKERAPPORT STATUS          0=GODKJ.  1=DRIFTFORS.  2= IKKE GODKJ.
LD TR0
AND<>(305) &1 C25_RAP_STATUS  ; VASKERAPPORT STATUS          0=GODKJ.  1=DRIFTFORS.  2= IKKE GODKJ.
@LD C25_STERIL_AVSLUTT  ; PAST23
LDNOT C25_STERILISER  ; PAST23
@AND C25_STERIL_OPPVARM  ; PAST23
ORLD
ANDLD
MOV(021) &0 C25_RAP_STATUS  ; VASKERAPPORT STATUS          0=GODKJ.  1=DRIFTFORS.  2= IKKE GODKJ.
LD TR0
ANDNOT C25_STERIL_AVSLUTT  ; PAST23
ANDNOT C25_SYRE_SKYLL  ; PAST23
TIM 0822 #10  ; P23_VASKER_AVBRUDD_S
LD TR0
AND C25_IND_VST80_K4  ; VASK PAST23
%LD C25_SYRE_SKYLL  ; PAST23
%LD C25_LUT_SKYLL  ; PAST23
ANDNOT C25_LUT_SYRE  ; PAST23
ORLD
ANDLD
OUT 964.10
LD TR0
LDNOT C25_STERIL_AVSLUTT  ; PAST23
AND 964.10
AND C25_STERIL_OPPVARM  ; PAST23
OR C25_STERIL_AVSLUTT  ; PAST23
%OR C25_STERIL_AVSLUTT  ; PAST23
ANDLD
SET C25_VASKERAPP_OK
LD TR0
ANDNOT P23_VASKER_AVBRUDD_S
%AND C25_IND_VST80_K4  ; VASK PAST23
ANDNOT C25_VASKERAPP_OK
ANDNOT P_On
MOV(021) #2 C25_RAP_STATUS  ; VASKERAPPORT STATUS          0=GODKJ.  1=DRIFTFORS.  2= IKKE GODKJ.
LD TR0
ANDNOT C25_IND_VST80_K4  ; VASK PAST23
AND P23_VASKER_AVBRUDD_S
RSET C25_VASKERAPP_OK
; rung 12: Ingen_kommentar_funnet

### Section VST80_K4_SIGNAL_N3

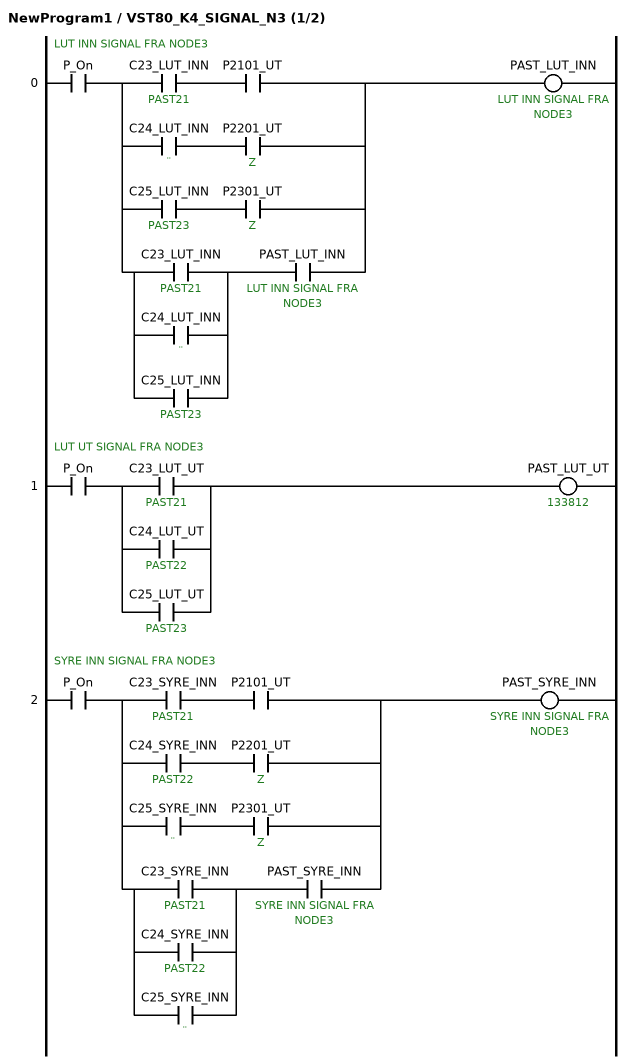
; rung 0: LUT INN SIGNAL FRA NODE3
LD P_On
LD C23_LUT_INN  ; PAST21
AND P2101_UT
LD C24_LUT_INN  ; ¨
AND P2201_UT  ; Z
ORLD
LD C25_LUT_INN  ; PAST23
AND P2301_UT  ; Z
ORLD
LD C23_LUT_INN  ; PAST21
OR C24_LUT_INN  ; ¨
OR C25_LUT_INN  ; PAST23
AND PAST_LUT_INN  ; LUT INN SIGNAL FRA NODE3
ORLD
ANDLD
OUT PAST_LUT_INN  ; LUT INN SIGNAL FRA NODE3
; rung 1: LUT UT SIGNAL FRA NODE3
LD P_On
LD C23_LUT_UT  ; PAST21
OR C24_LUT_UT  ; PAST22
OR C25_LUT_UT  ; PAST23
ANDLD
OUT PAST_LUT_UT  ; 133812
; rung 2: SYRE INN SIGNAL FRA NODE3
LD P_On
LD C23_SYRE_INN  ; PAST21
AND P2101_UT
LD C24_SYRE_INN  ; PAST22
AND P2201_UT  ; Z
ORLD
LD C25_SYRE_INN  ; ¨
AND P2301_UT  ; Z
ORLD
LD C23_SYRE_INN  ; PAST21
OR C24_SYRE_INN  ; PAST22
OR C25_SYRE_INN  ; ¨
AND PAST_SYRE_INN  ; SYRE INN SIGNAL FRA NODE3
ORLD
ANDLD
OUT PAST_SYRE_INN  ; SYRE INN SIGNAL FRA NODE3

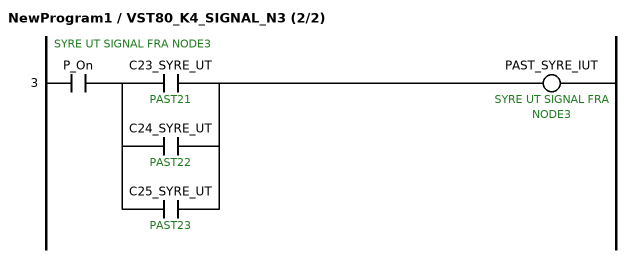
; rung 3: SYRE UT SIGNAL FRA NODE3
LD P_On
LD C23_SYRE_UT  ; PAST21
OR C24_SYRE_UT  ; PAST22
OR C25_SYRE_UT  ; PAST23
ANDLD
OUT PAST_SYRE_IUT  ; SYRE UT SIGNAL FRA NODE3
; rung 4: Ingen_kommentar_funnet

### Section VST80_K4_COND_OMSLAG

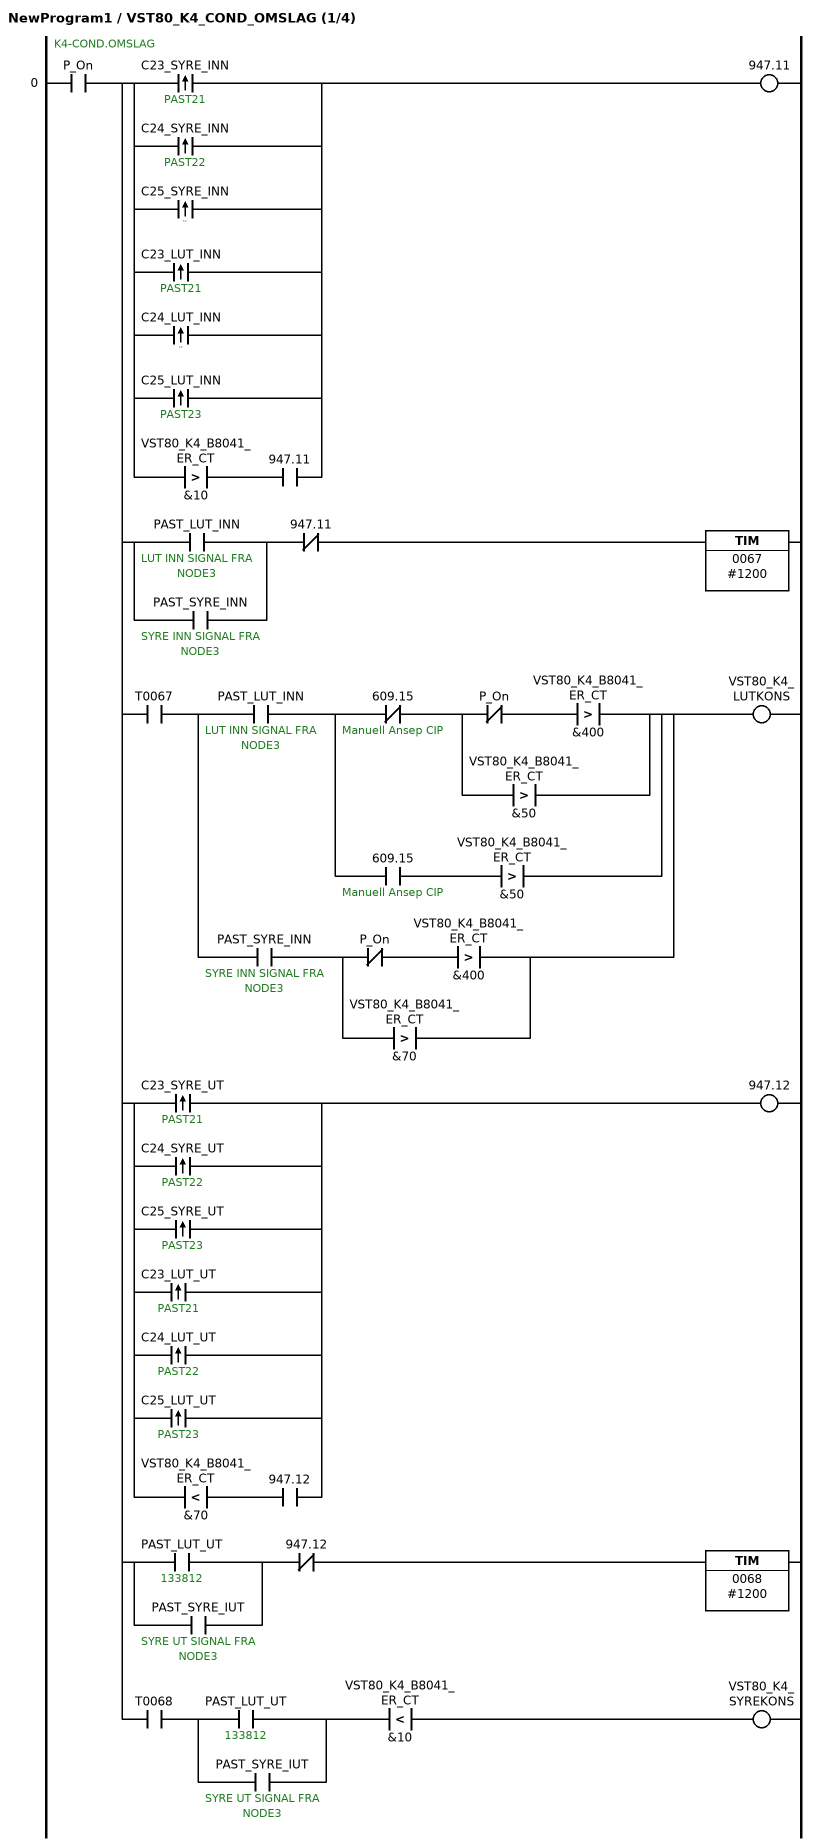
; rung 0: K4-COND.OMSLAG
LD P_On
OUT TR0
@LD C23_SYRE_INN  ; PAST21
@OR C24_SYRE_INN  ; PAST22
@OR C25_SYRE_INN  ; ¨
@OR C23_LUT_INN  ; PAST21
@OR C24_LUT_INN  ; ¨
@OR C25_LUT_INN  ; PAST23
LD>(320) VST80_K4_B8041_ER_CT &10
AND 947.11
ORLD
ANDLD
OUT 947.11
LD TR0
LD PAST_LUT_INN  ; LUT INN SIGNAL FRA NODE3
OR PAST_SYRE_INN  ; SYRE INN SIGNAL FRA NODE3
ANDLD
ANDNOT 947.11
TIM 0067 #1200
LD TR0
AND T0067
LD PAST_LUT_INN  ; LUT INN SIGNAL FRA NODE3
LDNOT 609.15  ; Manuell Ansep CIP
LDNOT P_On
AND>(320) VST80_K4_B8041_ER_CT &400
OR>(320) VST80_K4_B8041_ER_CT &50
ANDLD
LD 609.15  ; Manuell Ansep CIP
AND>(320) VST80_K4_B8041_ER_CT &50
ORLD
ANDLD
LD PAST_SYRE_INN  ; SYRE INN SIGNAL FRA NODE3
LDNOT P_On
AND>(320) VST80_K4_B8041_ER_CT &400
OR>(320) VST80_K4_B8041_ER_CT &70
ANDLD
ORLD
ANDLD
OUT VST80_K4_LUTKONS
LD TR0
@LD C23_SYRE_UT  ; PAST21
@OR C24_SYRE_UT  ; PAST22
@OR C25_SYRE_UT  ; PAST23
@OR C23_LUT_UT  ; PAST21
@OR C24_LUT_UT  ; PAST22
@OR C25_LUT_UT  ; PAST23
LD<(310) VST80_K4_B8041_ER_CT &70
AND 947.12
ORLD
ANDLD
OUT 947.12
LD TR0
LD PAST_LUT_UT  ; 133812
OR PAST_SYRE_IUT  ; SYRE UT SIGNAL FRA NODE3
ANDLD
ANDNOT 947.12
TIM 0068 #1200
LD TR0
AND T0068
LD PAST_LUT_UT  ; 133812
OR PAST_SYRE_IUT  ; SYRE UT SIGNAL FRA NODE3
ANDLD
AND<(310) VST80_K4_B8041_ER_CT &10
OUT VST80_K4_SYREKONS

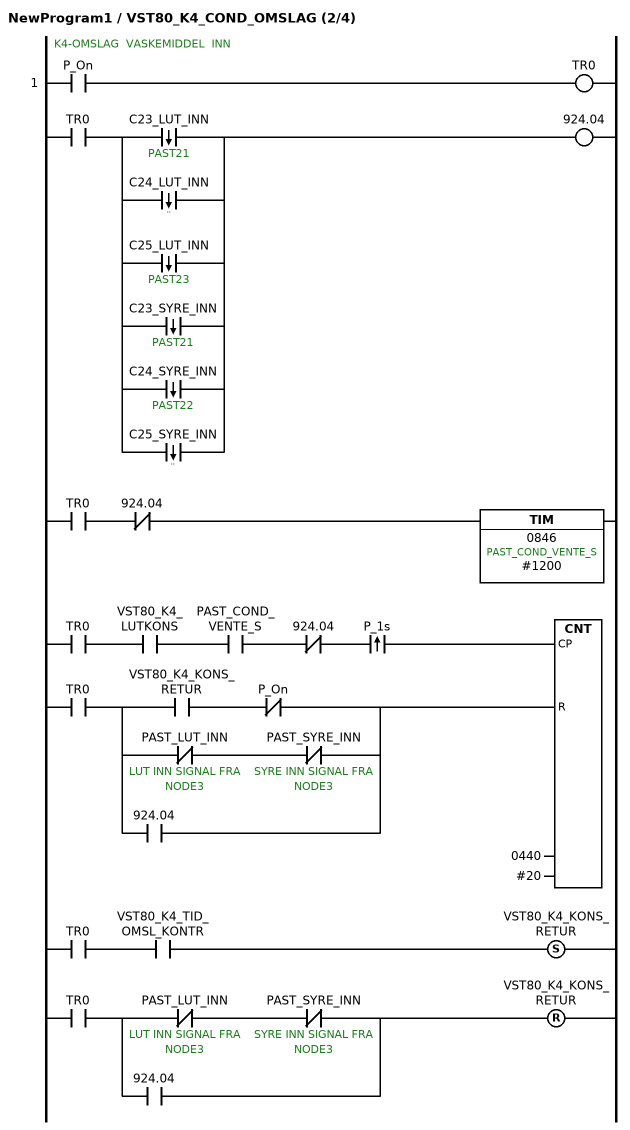
; rung 1: K4-OMSLAG  VASKEMIDDEL  INN
LD P_On
OUT TR0
%LD C23_LUT_INN  ; PAST21
%OR C24_LUT_INN  ; ¨
%OR C25_LUT_INN  ; PAST23
%OR C23_SYRE_INN  ; PAST21
%OR C24_SYRE_INN  ; PAST22
%OR C25_SYRE_INN  ; ¨
ANDLD
OUT 924.04
LD TR0
ANDNOT 924.04
TIM 0846 #1200  ; PAST_COND_VENTE_S
LD TR0
AND VST80_K4_LUTKONS
AND PAST_COND_VENTE_S
ANDNOT 924.04
@AND P_1s
LD TR0
LD VST80_K4_KONS_RETUR
ANDNOT P_On
LDNOT PAST_LUT_INN  ; LUT INN SIGNAL FRA NODE3
ANDNOT PAST_SYRE_INN  ; SYRE INN SIGNAL FRA NODE3
ORLD
OR 924.04
ANDLD
CNT 0440 #20
LD TR0
AND VST80_K4_TID_OMSL_KONTR
SET VST80_K4_KONS_RETUR
LD TR0
LDNOT PAST_LUT_INN  ; LUT INN SIGNAL FRA NODE3
ANDNOT PAST_SYRE_INN  ; SYRE INN SIGNAL FRA NODE3
OR 924.04
ANDLD
RSET VST80_K4_KONS_RETUR

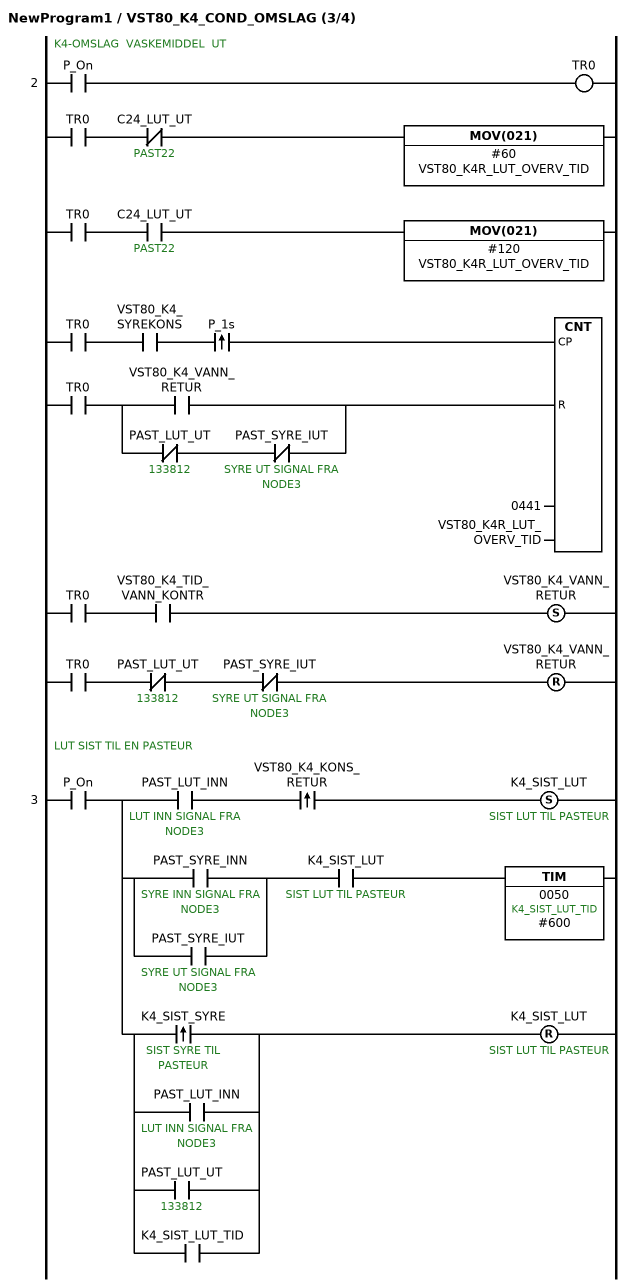
; rung 2: K4-OMSLAG  VASKEMIDDEL  UT
LD P_On
OUT TR0
ANDNOT C24_LUT_UT  ; PAST22
MOV(021) #60 VST80_K4R_LUT_OVERV_TID
LD TR0
AND C24_LUT_UT  ; PAST22
MOV(021) #120 VST80_K4R_LUT_OVERV_TID
LD TR0
AND VST80_K4_SYREKONS
@AND P_1s
LD TR0
LD VST80_K4_VANN_RETUR
LDNOT PAST_LUT_UT  ; 133812
ANDNOT PAST_SYRE_IUT  ; SYRE UT SIGNAL FRA NODE3
ORLD
ANDLD
CNT 0441 VST80_K4R_LUT_OVERV_TID
LD TR0
AND VST80_K4_TID_VANN_KONTR
SET VST80_K4_VANN_RETUR
LD TR0
ANDNOT PAST_LUT_UT  ; 133812
ANDNOT PAST_SYRE_IUT  ; SYRE UT SIGNAL FRA NODE3
RSET VST80_K4_VANN_RETUR
; rung 3: LUT SIST TIL EN PASTEUR
LD P_On
OUT TR0
AND PAST_LUT_INN  ; LUT INN SIGNAL FRA NODE3
@AND VST80_K4_KONS_RETUR
SET K4_SIST_LUT  ; SIST LUT TIL PASTEUR
LD TR0
LD PAST_SYRE_INN  ; SYRE INN SIGNAL FRA NODE3
OR PAST_SYRE_IUT  ; SYRE UT SIGNAL FRA NODE3
ANDLD
AND K4_SIST_LUT  ; SIST LUT TIL PASTEUR
TIM 0050 #600  ; K4_SIST_LUT_TID
LD TR0
@LD K4_SIST_SYRE  ; SIST SYRE TIL PASTEUR
OR PAST_LUT_INN  ; LUT INN SIGNAL FRA NODE3
OR PAST_LUT_UT  ; 133812
OR K4_SIST_LUT_TID
ANDLD
RSET K4_SIST_LUT  ; SIST LUT TIL PASTEUR

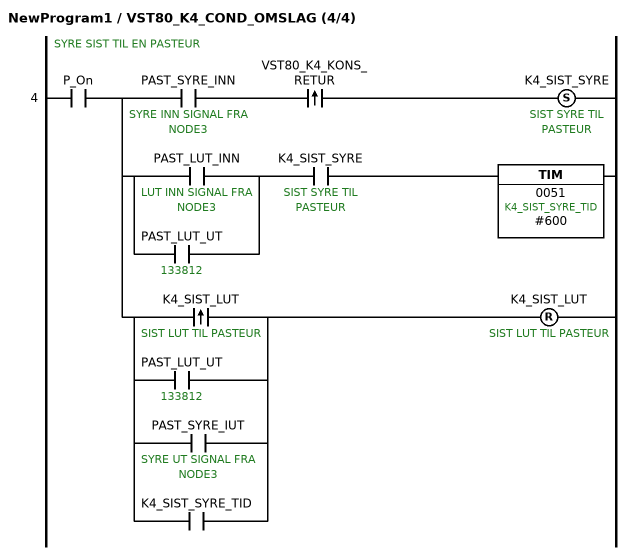
; rung 4: SYRE SIST TIL EN PASTEUR
LD P_On
OUT TR0
AND PAST_SYRE_INN  ; SYRE INN SIGNAL FRA NODE3
@AND VST80_K4_KONS_RETUR
SET K4_SIST_SYRE  ; SIST SYRE TIL PASTEUR
LD TR0
LD PAST_LUT_INN  ; LUT INN SIGNAL FRA NODE3
OR PAST_LUT_UT  ; 133812
ANDLD
AND K4_SIST_SYRE  ; SIST SYRE TIL PASTEUR
TIM 0051 #600  ; K4_SIST_SYRE_TID
LD TR0
@LD K4_SIST_LUT  ; SIST LUT TIL PASTEUR
OR PAST_LUT_UT  ; 133812
OR PAST_SYRE_IUT  ; SYRE UT SIGNAL FRA NODE3
OR K4_SIST_SYRE_TID
ANDLD
RSET K4_SIST_LUT  ; SIST LUT TIL PASTEUR
; rung 5: Ingen_kommentar_funnet

### Section VST80_K4_ANALOGSIGNAL_INN

